FUNCTION F_LogMessage : T_MaxString
VAR_INPUT
    Message : T_MaxString;
END_VAR

ADSLOGSTR(
    msgCtrlMask := ADSLOG_MSGTYPE_STRING OR ADSLOG_MSGTYPE_HINT OR ADSLOG_MSGTYPE_LOG,
    msgFmtStr := Message,
    strArg := '');

END_FUNCTION

(* stored: Version 1.1.0.1, ProductVersion 3.1.4024.3
   POU F_LogMessage: Id {a29b4cf0-9c7a-098b-1566-6f79e36b83d2}, SpecialFunc None *)
